# EPICS IOC start-up script: examples/test/PSI/AMI8000/AMI8121.iocsh
#- #############################################################################
#- mXsXXX naming
require ecmccfg AMI, "ECMC_VER=dev,NAMING=mXsXXX,EC_RATE=500"

#- #############################################################################
#- add slaves
${SCRIPTEXEC} ${ECMC_CONFIG_ROOT}addSlave.cmd, "HW_DESC=AMI8121"

epicsEnvSet("DRV_SLAVE", 0)
${SCRIPTEXEC} ${ECMC_CONFIG_ROOT}addAxisYaml.cmd, "FILE=cfg/AMI8121.yaml, ECMC_TMPDIR=/tmp/"
